RoboDK station: Controllernachricht.rdk

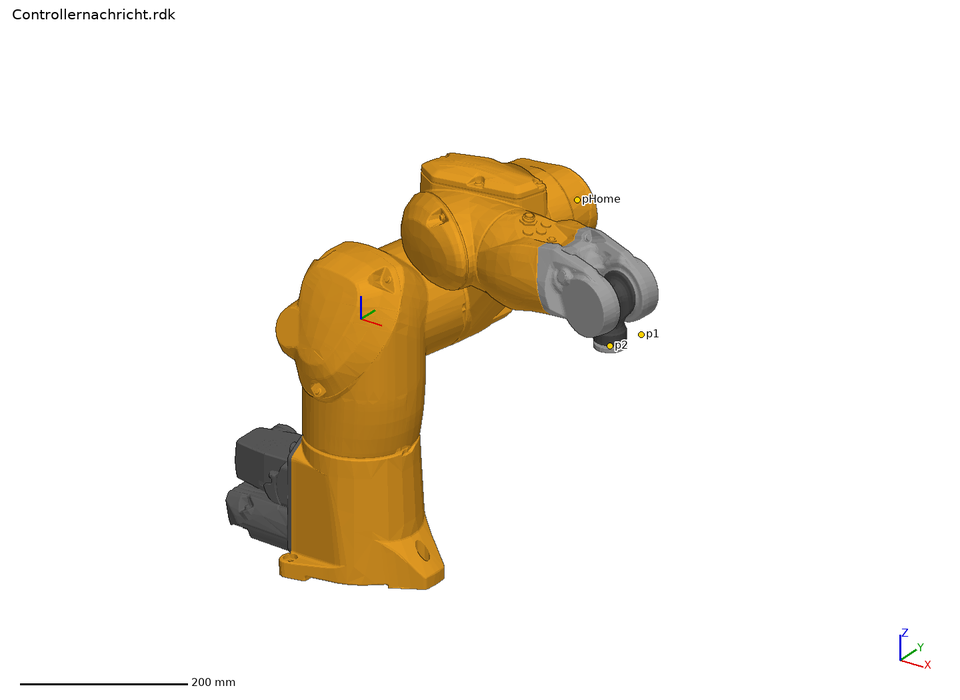
[picture v0: the station drawn from its stored meshes, robots at their saved joint values, targets as dots, program paths as lines]
Station Controllernachricht (saved by RoboDK 5.0.2). Poses are relative to the parent item; angles as X-Y-Z fixed-axis rotations.
  - frame Staubli TX2-40 Base at (0, 0, 320) mm
    - robot Staubli TX2-40: 6 axes, payload 1.7 kg, reach 515 mm, repeatability 0.02 mm, weight 29 kg
        modified DH rows (alpha deg, a mm, theta deg, d mm): 0, 0, 0, 320; -90, 0, -90, 35; 0, 225, -90, 0; -90, 0, 0, 225; 90, 0, 0, 0; -90, 0, 180, 65
        base shift (0, 0, -320) mm
        joint limits [-180, -125, -138, -270, -120, -270] to [180, 125, 138, 270, 133.5, 270]; home [0, 0, 90, 0, 0, 0]; saved at [-10.978, 47.352, 41.994, 0, 90.653, -10.978]
    - target pHome (Cartesian target) at (290, 35, 225) mm, rotated rx 0 ry 90 rz 0 deg; joints [0, 0, 90, 0, 0, 0] of Staubli TX2-40
    - target p1 (Cartesian target) at (380, 40, 70) mm, rotated rx 180 ry 0 rz -180 deg; joints [0.753, 44.255, 52.419, 0, 83.325, 0.753] of Staubli TX2-40
    - target p2 (Cartesian target) at (390, -40, 90) mm, rotated rx 180 ry 0 rz 180 deg; joints [-10.978, 47.352, 41.994, 0, 90.653, -10.978] of Staubli TX2-40
  - Python program Controllernachricht (listed below)

--- Python program Controllernachricht ---
# BEISPIELPROGRAMM: RTS-LIBRARY: CONTROLLERNACHRICHT ANZEIGEN.
# Führt 2 Bewegungen aus und gibt dann eine Nachricht einerseits
# in der Simulation, und andererseits auf dem Robotercontroller aus.

# Import der Librarys
from robolink import *
from robodk import *
from RTS import *

RDK = Robolink()

# Initialisierung aller Simulationsobjekte
rRobot = RDK.Item('Staubli TX2-40')
pHome = RDK.Item('pHome')
p1 = RDK.Item('p1')
p2 = RDK.Item('p2')


# Erstellen des RTS-Objektes. Falls im Programm kein Greifer genutzt wird, muss auch nicht zwingend einer übergeben werden.
RTS = RTS(RDK,rRobot)

# Führt 2 Bewegungen aus
rRobot.MoveJ(p1)
rRobot.MoveJ(p2)

# Gibt auf Controller und der Simulation die Nachricht "Nachricht1" aus.
RTS.boxAlert("Nachricht 1")

# Führt 2 Bewegungen aus
rRobot.MoveJ(p1)
rRobot.MoveJ(p2)

# Gibt auf Controller und der Simulation die Nachricht "Nachricht2" aus.
RTS.boxAlert("Nachricht 2")

# Führt 2 Bewegungen aus
rRobot.MoveJ(p1)
rRobot.MoveJ(p2)

# Gibt auf Controller und der Simulation die Nachricht "Programm ist fertig" aus.
RTS.boxAlert("Programm ist fertig")
